{attribute 'enable_dynamic_creation'}
FUNCTION_BLOCK FB_pHElectrodeCap EXTENDS FB_PieceBase
VAR_INPUT
END_VAR
VAR_OUTPUT
END_VAR
VAR
END_VAR

METHOD FB_init : BOOL
VAR_INPUT
	bInitRetains : BOOL; // if TRUE, the retain variables are initialized (warm start / cold start)
	bInCopyCode : BOOL;  // if TRUE, the instance afterwards gets moved into the copy code (online change)
END_VAR
eObjectType := E_ObjectType.OBJECTTYPE_pHElectrodeCap;
eObjectGroup := E_ObjectGroup.OBJECTGROUP_Piece;
END_METHOD

END_FUNCTION_BLOCK

(* stored: Version 1.1.0.1, ProductVersion 3.1.4022.18
   POU FB_pHElectrodeCap: Id {4a3f5242-be83-4670-a138-0118305bfb8a}, SpecialFunc None
   Method FB_init: Id {29d60f44-a8c7-42c3-8fbd-143ccb49c282} *)
